// TwinCAT 3 PLC project Template
// ProgramVersion: 3.1.4026.27
// CompilerDefines: VISU_USEPROPERTYINFO
// libraries:
//   [ApplicationBase], * (Beckhoff Automation LLC)
//   Tc2_Standard, * (Beckhoff Automation GmbH)
//   Tc2_System, * (Beckhoff Automation GmbH)
//   Tc3_PackML_V3, * (Beckhoff Automation GmbH)
// project tree:
//   / GlobalTextList.TcGTLO, MAIN.TcPOU, PlcTask.TcTTO
//   Machine/DUT/ ST_AxisRecipe.TcDUT, ST_Machine_HMI.TcDUT, ST_Recipe.TcDUT
//   Machine/Interface/ I_Machine.TcIO
//   Machine/ Machine.TcPOU, Machine_HMI.TcPOU
//   Visu/User Controls/ V_PackMLModule.TcVIS
//   Visu/ Visualization Manager.TcVMO (not stored), V_Main.TcVIS
// (motion and I/O tree: see PLC project unittests)
// real-time tasks:
//   TASK UnitTestsBase: cycle T#10ms, priority 20, ADS port 350
//   TASK VFFS: cycle T#10ms, priority 21, ADS port 351
//   TASK PlcTask: cycle T#10ms, priority 22, ADS port 352
//   TASK Job Task: cycle default, priority 32
//   TASK MC-Task (MET): cycle T#2ms, priority 3, ADS port 521
//   TASK MC-Task (MPT): cycle T#10ms, priority 9, ADS port 531
// variable links:

CONFIGURATION Template
    RESOURCE PLC ON TwinCAT3
        TASK PlcTask(INTERVAL := T#10ms, PRIORITY := 22);
        PROGRAM MAIN WITH PlcTask : MAIN;
    END_RESOURCE
END_CONFIGURATION

// ---- Machine/DUT/ST_AxisRecipe.TcDUT
TYPE ST_AxisRecipe :
	STRUCT
		Velocity	 : LREAL := 100;
		Acceleration : LREAL := 1000;
		Deceleration : LREAL := 1000;
		Jerk		 : LREAL := 1000;
	END_STRUCT
END_TYPE

// ---- Machine/DUT/ST_Machine_HMI.TcDUT
TYPE ST_Machine_HMI EXTENDS ST_HmiFunction :
	STRUCT
		Override : LREAL := 100.0;
	END_STRUCT
END_TYPE

// ---- Machine/DUT/ST_Recipe.TcDUT
TYPE ST_Recipe :
	STRUCT
		Axis : ST_AxisRecipe;
	END_STRUCT
END_TYPE

// ---- Machine/Interface/I_Machine.TcIO
INTERFACE I_Machine EXTENDS I_ContainStatemachine

PROPERTY Override : LREAL
SET
END_SET
END_PROPERTY

PROPERTY Recipe : REFERENCE TO ST_Recipe
GET
END_GET
END_PROPERTY

END_INTERFACE

// ---- MAIN.TcPOU
PROGRAM MAIN
VAR
	Machine : Machine('Machine');
END_VAR

IF NOT Machine.Initialized THEN
	Machine.Initialize();
	RETURN;
END_IF

Machine.CyclicLogic();

END_PROGRAM

// ---- Machine/Machine.TcPOU
FUNCTION_BLOCK Machine EXTENDS PackMLModule IMPLEMENTS I_Machine
VAR
	Events			  : TcEventClass('Machine');
	EventReactor	  : EventReactorPackMLVisitor('Event Reaction', THIS^);
	SyncedSquareWaves : SyncedSquareWaves('Waves');

	// Recipe
	_Recipe	   : ST_Recipe;
	RecipeFile : JsonFile<10000>('Recipe') := (Path := 'C:\Data\Recipe.json', SymbolName := 'Recipe', Datatype := 'ST_Recipe', nData := SIZEOF(_Recipe), pData := ADR(_Recipe));
END_VAR

VAR
	Machine_HMI : Machine_HMI('Machine', _Statemachine, THIS^);
END_VAR

VAR
	_Override : LREAL := 100.0;
END_VAR

METHOD Aborted : BOOL
END_METHOD

METHOD Aborting : BOOL
CASE SequenceState OF
	0:
		Aborting := TRUE;
END_CASE
END_METHOD

METHOD Clearing : BOOL
CASE SequenceState OF
	0:
		IF ResetComponents() AND ResetModules() THEN
			Clearing := TRUE;
		END_IF
END_CASE
END_METHOD

METHOD Execute : BOOL
END_METHOD

(*FB_Init is always available implicitly and it is used primarily for initialization.
The return value is not evaluated. For a specific influence, you can also declare the
methods explicitly and provide additional code there with the standard initialization
code. You can evaluate the return value.*)
METHOD FB_Init : BOOL
VAR_INPUT
	(* TRUE: the retain variables are initialized (reset warm / reset cold)*)
	bInitRetains	: BOOL;
	(* TRUE: the instance will be copied to the copy code afterward (online change)   *)
	bInCopyCode	: BOOL;
	Name	: ApplicationBase.T_MaxString;
END_VAR
Events.GenerateTcEvents(Name, ADR(TC_Events.Machine), SIZEOF(ST_Machine));
Events.RegisterWithParent(THIS^);
EventReactor.RegisterWithParent(THIS^);
Machine_HMI.RegisterWithParent(THIS^);
SyncedSquareWaves.RegisterWithParent(THIS^);

//
RecipeFile.RegisterWithParent(THIS^);
END_METHOD

(* This Module will be done initialize when ModuleInitialized := TRUE;, subequently all subitems will be called to be initialized *)
METHOD Initializing
VAR_INST
	UnitModeConfig : FB_PMLUnitModeConfig;
	SequenceState  : UDINT;
END_VAR
CASE SequenceState OF
	0:
		UnitModeConfig(eMode						  := E_PMLProtectedUnitMode.Production,
					   sName						  := 'Production',
					   bDisableClearing				  := FALSE,
					   bDisableStarting				  := FALSE,
					   bDisableSuspended			  := TRUE,
					   bDisableStopping				  := FALSE,
					   bDisableAborting				  := FALSE,
					   bDisableHolding				  := TRUE,
					   bDisableHeld					  := TRUE,
					   bDisableUnholding			  := TRUE,
					   bDisableSuspending			  := TRUE,
					   bDisableUnsuspending			  := TRUE,
					   bDisableResetting			  := TRUE,
					   bDisableIdle					  := TRUE,
					   bDisableCompleting			  := TRUE,
					   bDisableComplete				  := TRUE,
					   bEnableUnitModeChangeStopped	  := TRUE,
					   bEnableUnitModeChangeIdle	  := FALSE,
					   bEnableUnitModeChangeSuspended := FALSE,
					   bEnableUnitModeChangeExecute	  := FALSE,
					   bEnableUnitModeChangeAborted	  := TRUE,
					   bEnableUnitModeChangeHeld	  := FALSE,
					   bEnableUnitModeChangeComplete  := FALSE,
					   bError						  =>,
					   nErrorId						  =>);

		UnitModeConfig(eMode						  := E_PMLProtectedUnitMode.Manual,
					   sName						  := 'Manual',
					   bDisableClearing				  := FALSE,
					   bDisableStarting				  := FALSE,
					   bDisableSuspended			  := TRUE,
					   bDisableStopping				  := FALSE,
					   bDisableAborting				  := FALSE,
					   bDisableHolding				  := TRUE,
					   bDisableHeld					  := TRUE,
					   bDisableUnholding			  := TRUE,
					   bDisableSuspending			  := TRUE,
					   bDisableUnsuspending			  := TRUE,
					   bDisableResetting			  := TRUE,
					   bDisableIdle					  := TRUE,
					   bDisableCompleting			  := TRUE,
					   bDisableComplete				  := TRUE,
					   bEnableUnitModeChangeStopped	  := TRUE,
					   bEnableUnitModeChangeIdle	  := FALSE,
					   bEnableUnitModeChangeSuspended := FALSE,
					   bEnableUnitModeChangeExecute	  := FALSE,
					   bEnableUnitModeChangeAborted	  := TRUE,
					   bEnableUnitModeChangeHeld	  := FALSE,
					   bEnableUnitModeChangeComplete  := FALSE,
					   bError						  =>,
					   nErrorId						  =>);

		SequenceState := SequenceState + 10;

	10:
		RecipeFile.LoadFile();
		SequenceState := SequenceState + 10;

	20:
		IF NOT RecipeFile.Busy AND NOT RecipeFile.Error THEN
			RecipeFile.ReadSymbol();
			SequenceState := SequenceState + 10;
		END_IF

	30:
		ModuleInitialized := TRUE;
END_CASE

RecipeFile.CyclicLogic();
END_METHOD

METHOD OnCyclicCall
VAR_INST
	HmiEnableDisable : HmiEnableDisableAllVisitor;
	SetOverride		 : SetAllOverrideVisitor;
	EStopOK			 : BOOL;
END_VAR
IF _Statemachine.Mode.CurrentMode = E_PMLProtectedUnitMode.Manual THEN
	HmiEnableDisable.EnableHmi(THIS^);
ELSE
	HmiEnableDisable.DisableHmi(THIS^);
	Machine_HMI.Enable();
END_IF

//
SetOverride.Set(THIS^, _Override);
// Test Logic
IF NOT EStopOK THEN
	Events.RaiseEvent(E_Machine.EStop_Pressed);
END_IF
END_METHOD

PROPERTY Override : LREAL
SET
_Override := Override;
END_SET
END_PROPERTY

PROPERTY Recipe : REFERENCE TO ST_Recipe
GET
Recipe REF= _Recipe;
END_GET
END_PROPERTY

METHOD Starting : BOOL
CASE SequenceState OF
	0:
		Starting := TRUE;
END_CASE
END_METHOD

METHOD Stopped : BOOL
END_METHOD

METHOD Stopping : BOOL
CASE SequenceState OF
	0:
		Stopping := TRUE;
END_CASE
END_METHOD

END_FUNCTION_BLOCK

// ---- Machine/Machine_HMI.TcPOU
FUNCTION_BLOCK Machine_HMI EXTENDS PackMLStatemachine_HMI
VAR
	Machine : I_Machine;
	{ attribute 'TcHmiSymbol.AddSymbol' }
	{ attribute 'TcHmiSymbol.AddSymbol.UserGroups' := '__SystemAdministrators, Admin' }
	Machine_HMI : ST_Machine_HMI;
END_VAR

METHOD CyclicLogic
VAR_INST
	StartRT : R_TRIG;
	StopRT	: R_TRIG;
	ResetRT : R_TRIG;
END_VAR
IF Machine = 0 THEN
	RETURN;
END_IF

SUPER^.CyclicLogic();
Machine_HMI.Name	   := Name;
Machine_HMI.HmiEnabled := Enabled;
Machine.Override	   := Machine_HMI.Override;

// User buttons
Statemachine_HMI.StartPermissive := Statemachine_HMI.CurrentState = E_PMLState.Stopped;
Statemachine_HMI.StopPermissive	 := Statemachine_HMI.CurrentState <> E_PMLState.Aborted;
Statemachine_HMI.ResetPermissive := Statemachine_HMI.CurrentState = E_PMLState.Aborted;
StartRT(CLK := Statemachine_HMI.StartPressed);
IF StartRT.Q THEN
	Statemachine.ChangeState(E_PMLCommand.Start);
END_IF

StopRT(CLK := Statemachine_HMI.StopPressed);
IF StopRT.Q THEN
	IF Statemachine_HMI.CurrentState = E_PMLState.Stopped THEN
		Statemachine.ChangeState(E_PMLCommand.Abort);
	ELSE
		Statemachine.ChangeState(E_PMLCommand.Stop);
	END_IF
END_IF

ResetRT(CLK := Statemachine_HMI.ResetPressed);
IF ResetRT.Q THEN
	IF Statemachine_HMI.CurrentState = E_PMLState.Aborted THEN
		Statemachine.ChangeState(E_PMLCommand.Clear);
	ELSE
		Statemachine.ChangeState(E_PMLCommand.Reset);
	END_IF
END_IF
END_METHOD

(*FB_Init is always available implicitly and it is used primarily for initialization.
The return value is not evaluated. For a specific influence, you can also declare the
methods explicitly and provide additional code there with the standard initialization
code. You can evaluate the return value.*)
METHOD FB_Init : BOOL
VAR_INPUT
	(* TRUE: the retain variables are initialized (reset warm / reset cold)*)
	bInitRetains : BOOL;

	(* TRUE: the instance will be copied to the copy code afterward (online change)   *)
	bInCopyCode	 : BOOL;
	Name		 : ApplicationBase.T_MaxString;
	Statemachine : I_Statemachine;
	Machine		 : I_Machine;
END_VAR
THIS^.Machine := Machine;
END_METHOD

END_FUNCTION_BLOCK

// ---- GlobalTextList.TcGTLO
TEXTLIST GlobalTextList
  334 = '%s'
  874 = 'Abort'
  724 = 'Clear'
  690 = 'Complete'
  358 = 'Current Mode: %s'
  446 = 'Current State: %s'
  213 = 'Hold'
  75 = 'Maintenance'
  105 = 'Manual'
  648 = 'Production'
  96 = 'Reset'
  352 = 'Start'
  365 = 'Stop'
  732 = 'Suspend'
  152 = 'Unhold'
  225 = 'Unsuspend'
END_TEXTLIST

// ---- Visu/User Controls/V_PackMLModule.TcVIS
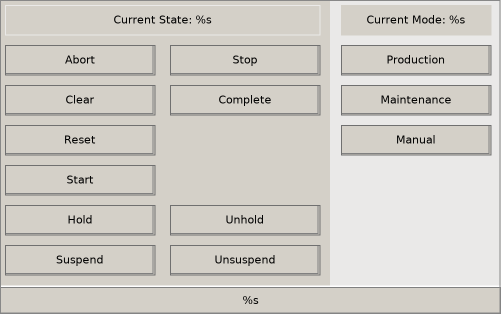
VISUALIZATION V_PackMLModule  // 501x314
VAR_IN_OUT
	PackML_HMI : ST_PackMLStatemachine_HMI;
END_VAR
    Rectangle (0,0 330x285)
    Textfield (5,5 315x30), "Current State: %s", text variable: PackML_HMI.CurrentState
    Button (5,45 150x30), "Abort"
        OnMouseClick: execute { PackML_HMI.StateCommand := E_PMLCommand.Abort; }
    Button (5,85 150x30), "Clear"
        OnMouseClick: execute { PackML_HMI.StateCommand := E_PMLCommand.Clear; }
    Button (5,125 150x30), "Reset"
        OnMouseClick: execute { PackML_HMI.StateCommand := E_PMLCommand.Reset; }
    Button (5,165 150x30), "Start"
        OnMouseClick: execute { PackML_HMI.StateCommand := E_PMLCommand.Start; }
    Button (170,85 150x30), "Complete"
        OnMouseClick: execute { PackML_HMI.StateCommand := E_PMLCommand.Complete; }
    Button (170,45 150x30), "Stop"
        OnMouseClick: execute { PackML_HMI.StateCommand := E_PMLCommand.Stop; }
    Button (5,205 150x30), "Hold"
        OnMouseClick: execute { PackML_HMI.StateCommand := E_PMLCommand.Hold; }
    Button (170,205 150x30), "Unhold"
        OnMouseClick: execute { PackML_HMI.StateCommand := E_PMLCommand.Unhold; }
    Button (5,245 150x30), "Suspend"
        OnMouseClick: execute { PackML_HMI.StateCommand := E_PMLCommand.Suspend; }
    Button (170,245 150x30), "Unsuspend"
        OnMouseClick: execute { PackML_HMI.StateCommand := E_PMLCommand.Unsuspend; }
    Rectangle (330,0 171x285)
    Textfield (341,5 150x30), "Current Mode: %s", text variable: PackML_HMI.CurrentMode
    Button (341,45 150x30), "Production"
        OnMouseClick: execute { PackML_HMI.ModeCommand := 1; }
    Button (341,85 150x30), "Maintenance"
        OnMouseClick: execute { PackML_HMI.ModeCommand := 2; }
    Button (341,125 150x30), "Manual"
        OnMouseClick: execute { PackML_HMI.ModeCommand := 3; }
    Textfield (0,287 501x27), "%s", text variable: PackML_HMI.Name
END_VISUALIZATION

// ---- Visu/V_Main.TcVIS
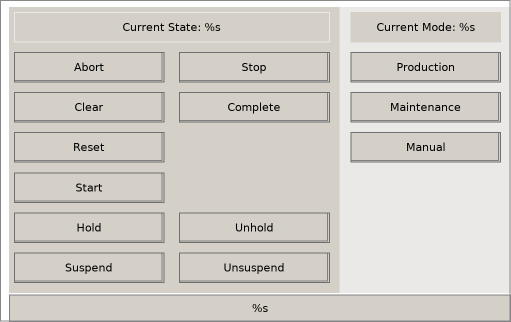
VISUALIZATION V_Main  // 511x322
    Frame (9,7 502x315)
        shows V_PackMLModule(PackML_HMI := MAIN.Machine.Machine_HMI.Statemachine_HMI)
END_VISUALIZATION
